FUNCTION_BLOCK sequence_T_08_ADAPTER (* Composite wrapper around sequence_T_08: Event/BOOL outputs bundled into AX/AS adapters, DT_Sx_Sy times each fed via its own ATM adapter socket. timeOut stays internal, not exposed. *)
  (* Standard: 61499-2; Description: Copyright (c) 2026 HR Agrartechnik GmbH This program and the accompanying materials are made available under the terms of the Eclipse Public License 2.0 which is available at https://www.eclipse.org/legal/epl-2.0/ SPDX-License-Identifier: EPL-2.0 *)
  (* Version 1.0, 2026-08-14, Franz Höpfinger, HR Agrartechnik GmbH, initial API and implementation *)
  PACKAGE logiBUS::utils::sequence::timed;
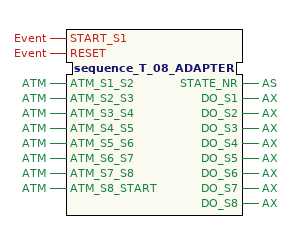
  EVENT_INPUT
    START_S1; (* jump from START to State_01 *)
    RESET; (* Reset from any State to START *)
  END_EVENT
  SOCKETS
    ATM_S1_S2 : adapter::types::unidirectional::ATM; (* State_01 to State_02 timed *)
    ATM_S2_S3 : adapter::types::unidirectional::ATM; (* State_02 to State_03 timed *)
    ATM_S3_S4 : adapter::types::unidirectional::ATM; (* State_03 to State_04 timed *)
    ATM_S4_S5 : adapter::types::unidirectional::ATM; (* State_04 to State_05 timed *)
    ATM_S5_S6 : adapter::types::unidirectional::ATM; (* State_05 to State_06 timed *)
    ATM_S6_S7 : adapter::types::unidirectional::ATM; (* State_06 to State_07 timed *)
    ATM_S7_S8 : adapter::types::unidirectional::ATM; (* State_07 to State_08 timed *)
    ATM_S8_START : adapter::types::unidirectional::ATM; (* State_08 to START timed *)
  END_SOCKETS
  PLUGS
    STATE_NR : adapter::types::unidirectional::AS; (* State Number Adapter *)
    DO_S1 : adapter::types::unidirectional::AX; (* Output if State_01 is active *)
    DO_S2 : adapter::types::unidirectional::AX; (* Output if State_02 is active *)
    DO_S3 : adapter::types::unidirectional::AX; (* Output if State_03 is active *)
    DO_S4 : adapter::types::unidirectional::AX; (* Output if State_04 is active *)
    DO_S5 : adapter::types::unidirectional::AX; (* Output if State_05 is active *)
    DO_S6 : adapter::types::unidirectional::AX; (* Output if State_06 is active *)
    DO_S7 : adapter::types::unidirectional::AX; (* Output if State_07 is active *)
    DO_S8 : adapter::types::unidirectional::AX; (* Output if State_08 is active *)
  END_PLUGS
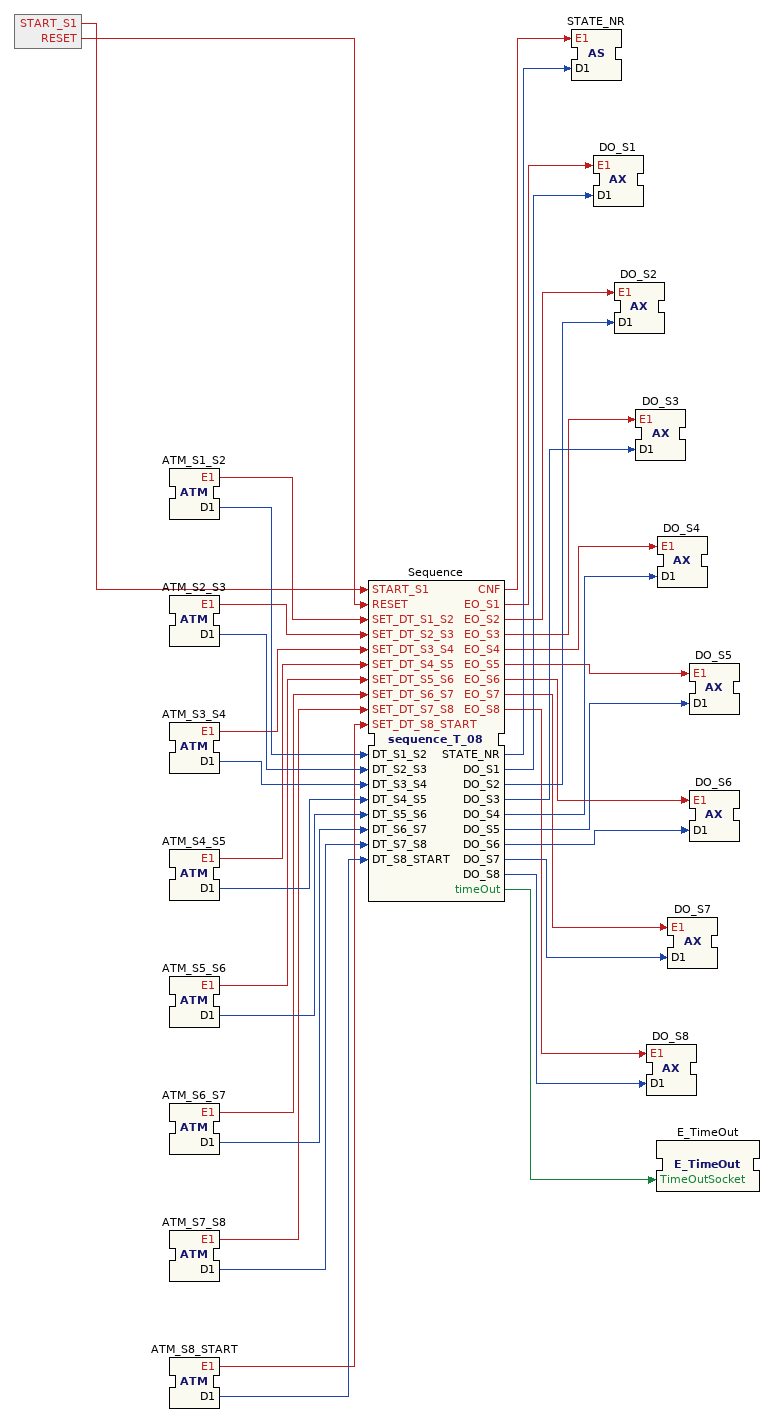
  FBS
    Sequence : logiBUS::utils::sequence::timed::sequence_T_08;
    E_TimeOut : iec61499::events::E_TimeOut;
  END_FBS
  EVENT_CONNECTIONS
    START_S1 TO Sequence.START_S1;
    RESET TO Sequence.RESET;
    ATM_S1_S2.E1 TO Sequence.SET_DT_S1_S2;
    ATM_S2_S3.E1 TO Sequence.SET_DT_S2_S3;
    ATM_S3_S4.E1 TO Sequence.SET_DT_S3_S4;
    ATM_S4_S5.E1 TO Sequence.SET_DT_S4_S5;
    ATM_S5_S6.E1 TO Sequence.SET_DT_S5_S6;
    ATM_S6_S7.E1 TO Sequence.SET_DT_S6_S7;
    ATM_S7_S8.E1 TO Sequence.SET_DT_S7_S8;
    ATM_S8_START.E1 TO Sequence.SET_DT_S8_START;
    Sequence.CNF TO STATE_NR.E1;
    Sequence.EO_S1 TO DO_S1.E1;
    Sequence.EO_S2 TO DO_S2.E1;
    Sequence.EO_S3 TO DO_S3.E1;
    Sequence.EO_S4 TO DO_S4.E1;
    Sequence.EO_S5 TO DO_S5.E1;
    Sequence.EO_S6 TO DO_S6.E1;
    Sequence.EO_S7 TO DO_S7.E1;
    Sequence.EO_S8 TO DO_S8.E1;
  END_CONNECTIONS
  DATA_CONNECTIONS
    ATM_S1_S2.D1 TO Sequence.DT_S1_S2;
    ATM_S2_S3.D1 TO Sequence.DT_S2_S3;
    ATM_S3_S4.D1 TO Sequence.DT_S3_S4;
    ATM_S4_S5.D1 TO Sequence.DT_S4_S5;
    ATM_S5_S6.D1 TO Sequence.DT_S5_S6;
    ATM_S6_S7.D1 TO Sequence.DT_S6_S7;
    ATM_S7_S8.D1 TO Sequence.DT_S7_S8;
    ATM_S8_START.D1 TO Sequence.DT_S8_START;
    Sequence.STATE_NR TO STATE_NR.D1;
    Sequence.DO_S1 TO DO_S1.D1;
    Sequence.DO_S2 TO DO_S2.D1;
    Sequence.DO_S3 TO DO_S3.D1;
    Sequence.DO_S4 TO DO_S4.D1;
    Sequence.DO_S5 TO DO_S5.D1;
    Sequence.DO_S6 TO DO_S6.D1;
    Sequence.DO_S7 TO DO_S7.D1;
    Sequence.DO_S8 TO DO_S8.D1;
  END_CONNECTIONS
  ADAPTER_CONNECTIONS
    Sequence.timeOut TO E_TimeOut.TimeOutSocket;
  END_CONNECTIONS
END_FUNCTION_BLOCK
